{attribute 'qualified_only'}
VAR_GLOBAL PERSISTENT
	Tags: CTH_LA02;
END_VAR

(* stored: Version 1.1.0.1, ProductVersion 3.1.4024.6
   GVL ADS_CTH: Id {7c476450-b4d3-4481-ba09-185ae0de07d1} *)
